SUBAPPLICATION Ventilsteuerung_Uebung_071b (* WBSD auf UT ausgeben, Q1 Schalten wenn Speed >0 *)
  (* Standard: 61499-2 *)
  (* Version 1.0, 2023-10-23, franz *)
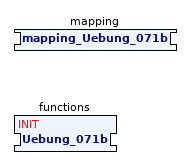
  SUBAPPS
    mapping : mapping_Uebung_071b;
    functions : Uebung_071b;
  END_SUBAPPS
END_SUBAPPLICATION
